// TIA Portal V19 export
FUNCTION_BLOCK "TYPIC_C215_IF_PBK"   // FB128, FBD
{ S7_Optimized_Access := 'TRUE' }
AUTHOR : OCOTECH
FAMILY : Typical
NAME : C215.703
// stored: MemoryReserve 10, SetENOAutomatically false
   VAR_INPUT
      EXT_AUT { ExternalAccessible := 'False'; ExternalVisible := 'False'; ExternalWritable := 'False'} : Bool;   // Externe (hoofd) beveiliging (1 = OK)
      EXT_HW { ExternalAccessible := 'False'; ExternalVisible := 'False'; ExternalWritable := 'False'} : Bool;   // Sturings hardware (PLC) bewaking (1 = OK)
      IN_AUT_C215 { ExternalAccessible := 'False'; ExternalVisible := 'False'; ExternalWritable := 'False'} : Bool;   // Serie geschakelde beveiligingen (1 = OK)
      IN_BAT { ExternalAccessible := 'False'; ExternalVisible := 'False'; ExternalWritable := 'False'} : Bool;   // Batterij (1 = OK)
   END_VAR
   VAR_OUTPUT
      VAR_IF_PBK { ExternalAccessible := 'False'; ExternalVisible := 'False'; ExternalWritable := 'False'} : "C215_VAR_IF_PBK_TYPIC";   // Struct met alle variabelen naar bovenliggende functies
   END_VAR
   VAR
      STO { ExternalWritable := 'False'} : Struct   // Storingen
         A001 : Bool;   // Beveiliging aangesproken
         A002 : Bool;   // Storing batterij
      END_STRUCT;
      VAR { ExternalWritable := 'False'} : Struct   // Variabelen
         EXT_AUT { ExternalAccessible := 'False'; ExternalVisible := 'False'} : Bool;   // Externe (hoofd) beveiliging aangesproken
         EXT_HW { ExternalAccessible := 'False'; ExternalVisible := 'False'} : Bool;   // Sturings hardware (PLC) in storing
      END_STRUCT;
   END_VAR
BEGIN
END_FUNCTION_BLOCK
